// TIA Portal V17 export
// export: Created 2022-07-28T18:03:03.762055Z, ExportSetting None, DisplayName Totally Integrated Automation Portal, DisplayVersion V17, DisplayName TIA Portal Openness, DisplayVersion V17, DisplayName TIA Portal Teamcenter Gateway, DisplayVersion V17, DisplayName TIA Portal Version Control Interface, DisplayVersion V17, DisplayName TIA Portal Test Suite Advanced, DisplayVersion V17, DisplayName SINAMICS Startdrive Advanced, DisplayVersion V17, DisplayName SINAMICS DCC, DisplayVersion V17, DisplayName SINAMICS Startdrive G130, G150, S120, S150, SINAMICS MV, S210, DisplayVersion V17, DisplayName SINAMICS Startdrive G110M, G120, G120C, G120D, G120P, G115D, DisplayVersion V17, DisplayName STEP 7 Professional, DisplayVersion V17, DisplayName SIMATIC Energy Suite, DisplayVersion V17, DisplayName STEP 7 CFC, DisplayVersion V17, DisplayName STEP 7 Safety, DisplayVersion V17, DisplayName WinCC Advanced / Unified PC, DisplayVersion V17, DisplayName SIMATIC Visualization Architect, DisplayVersion V17
DATA_BLOCK "D_Filter_LTR46_LT1"   // DB11
AUTHOR : VS
FAMILY : Simulation
VERSION : 2.0
// stored: InstanceOfName Lib_FB_PT1_Ramp, InstanceOfType FB
"Lib_FB_PT1_Ramp"
   // VAR_INPUT
   //    i_Reset : Bool;
   //    i_Invert : Bool;
   //    ir_Input : Real;
   //    ir_T1_sec : Real;
   //    ir_K : Real;
   //    ir_T_cycle_sec : Real;
   //    ir_OffSet_Out : Real;
   //    ir_Delta : Real;
   // END_VAR
   // VAR_OUTPUT
   //    q_DataErr : Bool;
   //    qr_Output : Real;
   // END_VAR
   // VAR
   //    s_FirstCall : Bool;
   //    sr_Output : Real;
   //    sr_T1_sec_Old : Real;
   //    sr_K_Old : Real;
   //    sr_T_cycle_sec_Old : Real;
   //    sr_InPart : Real;
   //    sr_ExpPart : Real;
   // END_VAR
BEGIN
END_DATA_BLOCK
